PROGRAM MAIN
VAR
	MC_ReadActualVelocity: MC_ReadActualVelocity;
	state: state;
	
	reset_output:ST_McOutputs;
	axis_Reset: MC_Reset;
	ReadP_Valid:BOOL;
	ReadV_Valid:BOOL;
	power1: MC_Power;
	
	power1_output:ST_McOutputs;
	
    axis: AXIS_REF;
	StartInit: BOOL := 1;
	MC_MoveVelocity_0: MC_MoveVelocity;
	
	MoveVelocity_output:ST_McOutputs;
	MC_MoveVelocity_1: MC_MoveVelocity;
	MC_ReadActualPosition: MC_ReadActualPosition;
END_VAR

// Programmablauf mittels Zustandsautomat
CASE state OF
	
	INIT:
		MC_MoveVelocity_0.Execute := FALSE;
		Power1.Enable:=FALSE;
		axis_Reset.Execute := FALSE;
		state := POWER_ON;
		
	POWER_ON:
		Power1.Enable := TRUE;
		IF power1.Status THEN
				state := MOVE_ON;
		ELSIF power1.Error THEN
				state := ERROR;
		END_IF

	MOVE_ON:
		
		IF GVL.PID_Output>=0 THEN
			MC_MoveVelocity_0.Direction := MC_Positive_Direction;
			GVL.Velocity := GVL.PID_Output;
		ELSIF GVL.PID_Output<0 THEN
			MC_MoveVelocity_0.Direction := MC_Negative_Direction;
			GVL.Velocity := (-1) * GVL.PID_Output;
		ELSE MC_MoveVelocity_0.Direction := MC_Undefined_Direction;
		END_IF

		
		MC_MoveVelocity_0.Execute := TRUE;
		IF MoveVelocity_output.Done THEN
			MC_MoveVelocity_0.Execute := FALSE;
			state := MOVE_ON;
		ELSIF MC_MoveVelocity_0.CommandAborted OR MC_MoveVelocity_0.Error THEN
			state := ERROR;
		END_IF
		
	ERROR:
		IF axis.Status.Error THEN
			state := P_RESET;	(* axis error requires reset *)
		ELSE
			state := INIT;		(* function block errors don't need a reset *)
		END_IF
		
	P_RESET:
		axis_Reset.Execute := TRUE;
		MC_MoveVelocity_0.Execute := FALSE;
		IF axis_Reset.Done  THEN
			state := INIT;
		ELSIF axis_Reset.Error  THEN
			state := INIT; 
		END_IF
END_CASE

axis();
Power();
ActMove();
ReadP_V();
Reset();

ACTION ActMove:
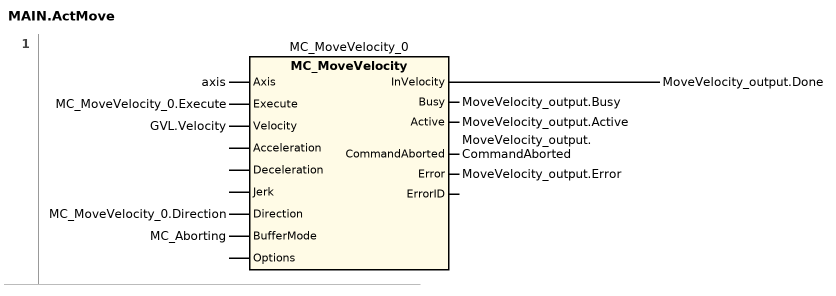
// NETWORK 1
MC_MoveVelocity_0(
    Axis := axis,
    Execute := MC_MoveVelocity_0.Execute,
    Velocity := GVL.Velocity,
    Direction := MC_MoveVelocity_0.Direction,
    BufferMode := MC_Aborting,
    Busy => MoveVelocity_output.Busy,
    Active => MoveVelocity_output.Active,
    CommandAborted => MoveVelocity_output.CommandAborted,
    Error => MoveVelocity_output.Error); // MC_MoveVelocity
MoveVelocity_output.Done := MC_MoveVelocity_0.InVelocity;
END_ACTION

ACTION Power:
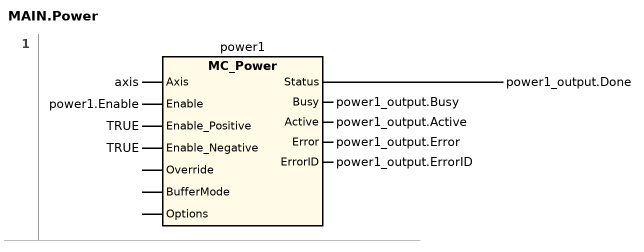
// NETWORK 1
power1(
    Axis := axis,
    Enable := power1.Enable,
    Enable_Positive := TRUE,
    Enable_Negative := TRUE,
    Busy => power1_output.Busy,
    Active => power1_output.Active,
    Error => power1_output.Error,
    ErrorID => power1_output.ErrorID); // MC_Power
power1_output.Done := power1.Status;
END_ACTION

ACTION ReadP_V:
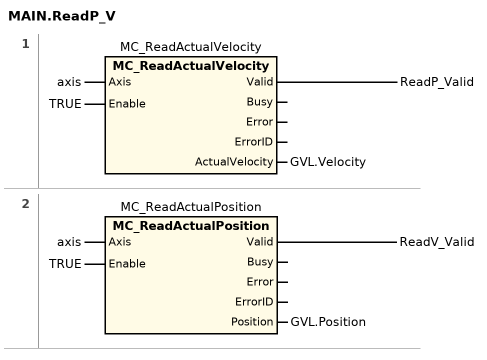
// NETWORK 1
MC_ReadActualVelocity(Axis := axis, Enable := TRUE, ActualVelocity => GVL.Velocity);
ReadP_Valid := MC_ReadActualVelocity.Valid;

// NETWORK 2
MC_ReadActualPosition(Axis := axis, Enable := TRUE, Position => GVL.Position);
ReadV_Valid := MC_ReadActualPosition.Valid;
END_ACTION

ACTION Reset:
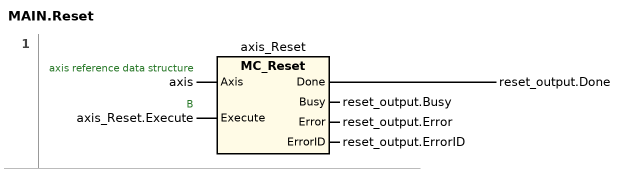
// NETWORK 1
//   axis: axis reference data structure
//   axis_Reset.Execute: B
axis_Reset(
    Axis := axis,
    Execute := axis_Reset.Execute,
    Busy => reset_output.Busy,
    Error => reset_output.Error,
    ErrorID => reset_output.ErrorID); // MC_Reset
reset_output.Done := axis_Reset.Done;
END_ACTION

END_PROGRAM

(* stored: Version 1.1.0.1, ProductVersion 3.1.4024.9
   POU MAIN: Id {534445fb-a9af-45c0-84b6-2e30f7c91eb2}, SpecialFunc None
   Action ActMove: Id {7c7f73c4-4ac9-4f89-b369-ff84303573f9}
   Action Power: Id {8b469144-5c09-487e-8637-7d166d37593e}
   Action ReadP_V: Id {4fb1b366-fac7-45a0-822a-d6e5a92b9fcd}
   Action Reset: Id {d4c531c5-ab2c-485e-947c-8ec7bbf86e8a} *)
